{attribute addProperty BoxType "ELM2642-0000-0016"}
{attribute addProperty Id "Outputs_Channel_2AT %Q*Outputs_Channel_E6FE5E20162"}
{attribute addProperty CRC "451447974"}
{attribute addProperty SizeInBites "16"}
{attribute addProperty SizeInBytes "2"}
TYPE DO_Group_2_Outputs_1AE88CA6 :
STRUCT
	{attribute addProperty Name "Outputs_Channel_2"}
	Outputs_Channel_2 AT %Q* : Outputs_Channel_E6FE5E20;
END_STRUCT
END_TYPE

(* stored: Version 1.2.0.0, ProductVersion 3.1.4024.9
   DUT DO_Group_2_Outputs_1AE88CA6: Id {554672f6-c345-42ba-9be0-5128adca8aa9} *)
